(* IEC 61131-3 sources: plc_programming/Ejercicios/Casos de estudio/Ejemplo_01/build, 2 files *)

(* ---- plc.st ---- *)
TYPE
  LOGLEVEL : (CRITICAL, WARNING, INFO, DEBUG) := INFO;
END_TYPE

FUNCTION_BLOCK LOGGER
  VAR_INPUT
    TRIG : BOOL;
    MSG : STRING;
    LEVEL : LOGLEVEL := INFO;
  END_VAR
  VAR
    TRIG0 : BOOL;
  END_VAR

  IF TRIG AND NOT TRIG0 THEN
  {{
   LogMessage(GetFbVar(LEVEL),(char*)GetFbVar(MSG, .body),GetFbVar(MSG, .len));
  }}
  END_IF;
  TRIG0:=TRIG;
END_FUNCTION_BLOCK

PROGRAM EP1
  VAR
    Start1 : BOOL;
    Stop1 : BOOL;
    Motor1 : BOOL;
    Start2 : BOOL;
    Stop2 : BOOL;
    Motor2 : BOOL;
    L1 : BOOL;
    L2 : BOOL;
  END_VAR

  Motor1 := NOT(Stop1) AND (Motor1 OR Start1);
  Motor2 := NOT(Stop2) AND (Motor2 OR Start2);
  L1 := Motor2 AND Motor1;
  L2 := NOT(L1) AND (Motor1 OR Motor2);
END_PROGRAM

CONFIGURATION Config0

  RESOURCE Res0 ON PLC
    TASK task0(INTERVAL := T#20ms,PRIORITY := 0);
    PROGRAM instance0 WITH task0 : EP1;
  END_RESOURCE
END_CONFIGURATION

(* ---- generated_plc.st ---- *)
PROGRAM EP1
  VAR
    Start1 : BOOL;
    Stop1 : BOOL;
    Motor1 : BOOL;
    Start2 : BOOL;
    Stop2 : BOOL;
    Motor2 : BOOL;
    L1 : BOOL;
    L2 : BOOL;
  END_VAR

  Motor1 := NOT(Stop1) AND (Motor1 OR Start1);
  Motor2 := NOT(Stop2) AND (Motor2 OR Start2);
  L1 := Motor2 AND Motor1;
  L2 := NOT(L1) AND (Motor1 OR Motor2);
END_PROGRAM

CONFIGURATION Config0

  RESOURCE Res0 ON PLC
    TASK task0(INTERVAL := T#20ms,PRIORITY := 0);
    PROGRAM instance0 WITH task0 : EP1;
  END_RESOURCE
END_CONFIGURATION
